// TIA Portal V16 export
// export: Created 2023-08-28T09:37:54.0618046Z, ExportSetting WithDefaults, DisplayName Totally Integrated Automation Portal, DisplayVersion V16 Update 6, DisplayName TIA Portal Version Control Interface, DisplayVersion V16 Update 2, DisplayName TIA Portal Openness, DisplayVersion V16 Update 6, DisplayName STEP 7 Professional, DisplayVersion V16 Update 6, DisplayName STEP 7 Safety, DisplayVersion V16, DisplayName WinCC Advanced, DisplayVersion V16 Update 6
VAR_GLOBAL   // PLC tag table "PID"
   switc_manualPID AT %M206.5 : Bool;   // Przełacznik regulator PID na manualne zadawanie
   setUPbar AT %M300.3 : Bool;   // Znacznik generatora czasowego podnoszenia wartości zadanej ciśnienia
   setDownbar AT %M300.4 : Bool;   // Znacznik generatora czasowego obniżania wartości ciśnienia
   enableAutomaticPIDreset AT %M300.7 : Bool;   // Znacznik automatycznego wykonania resetu PID
   lastError AT %MD301 : DWord;   // ostatni błąd
   stateBeforeError AT %MW305 : Int;   // bufor ostatnich błędów
   ResetPIDManual AT %M1100.0 : Bool;   // Ręczny reset PID
   Reset_PID1 AT %M14.4 : Bool;   // Znacznik resetu PID1
END_VAR
